FUNCTION_BLOCK TEMPLATE_BASICFB
  (* Standard: 61499-2 *)
  (* Version 1.0, 11-01-12, GASR, Universidade do Estado de Santa Catarina *)
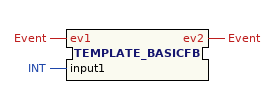
  EVENT_INPUT
    ev1;
  END_EVENT
  EVENT_OUTPUT
    ev2;
  END_EVENT
  VAR_INPUT
    input1 : INT;
  END_VAR
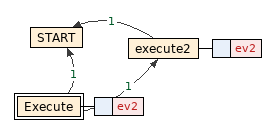
  EC_STATES
    Execute : -> ev2;
    START;
    execute2 : -> ev2;
  END_STATES
  EC_TRANSITIONS
    Execute TO START := 1;
    Execute TO execute2 := 1;
    execute2 TO START := 1;
  END_TRANSITIONS
END_FUNCTION_BLOCK
